FUNCTION_BLOCK ABSTRACT A_ContinuousDrive //generic drive that can only traverse in either direction or stop
VAR_INPUT
	bEnable : BOOL;
END_VAR
VAR_OUTPUT
	contact AT %I* : BOOL;
	
	outerLimit AT %I* : BOOL; //SMC sliders do not use this
	home AT %I* : BOOL;
	innerLimit AT %I* : BOOL;
	
	homeSet : BOOL;
	busy : BOOL;
	error : BOOL;
END_VAR
VAR
	step : Homing;
END_VAR

METHOD ABSTRACT homingSequence : BOOL
VAR_INPUT
END_VAR
END_METHOD

METHOD ABSTRACT moveContinuous : BOOL
VAR_INPUT
	direction : MC_Direction;
END_VAR
END_METHOD

METHOD ABSTRACT stop : BOOL
VAR_INPUT
END_VAR
END_METHOD

END_FUNCTION_BLOCK

(* stored: Version 1.1.0.1, ProductVersion 3.1.4024.11
   POU A_ContinuousDrive: Id {0abc7204-321d-448b-a2d6-f81a2f9d40da}, SpecialFunc None
   Method homingSequence: Id {aeec6ab2-d9e1-4729-85e6-30d35385fa84}
   Method moveContinuous: Id {5dab9c49-79fc-4eda-ae89-86f7ebf23aa2}
   Method stop: Id {3650c7e9-87dd-4a3a-8c61-5eec42a10cce} *)
